// Mitsubishi GX Works2 project: part_B_group31   PLC: FX3G

// global labels: Global1
VAR_GLOBAL
  Ac_start AT X007 : BOOL;
  Ac_stop AT X005 : BOOL;
  Ac_keepOn AT M0 : BOOL;
  one_hour AT TC6 : BOOL;
END_VAR
VAR_GLOBAL CONSTANT
  const_1hour : INT := 60;
END_VAR
VAR_GLOBAL
  one_hour_VAL AT TS6 : BOOL;
  sen_move AT X001 : BOOL;
  Last_move AT M1 : BOOL;
  sen_window AT X002 : BOOL;
  Ac_on AT Y001 : BOOL;
  check_move AT M4 : BOOL;
  Alarm AT Y002 : BOOL;
END_VAR

// task Task_01 (event TRUE, interval 0, priority 31): POU_01

PROGRAM POU_01
(* structured ladder/FBD written out as ST: instructions are called as NAME(EN, inputs, outputs); _pN, _eN, _tN stand for wires *)
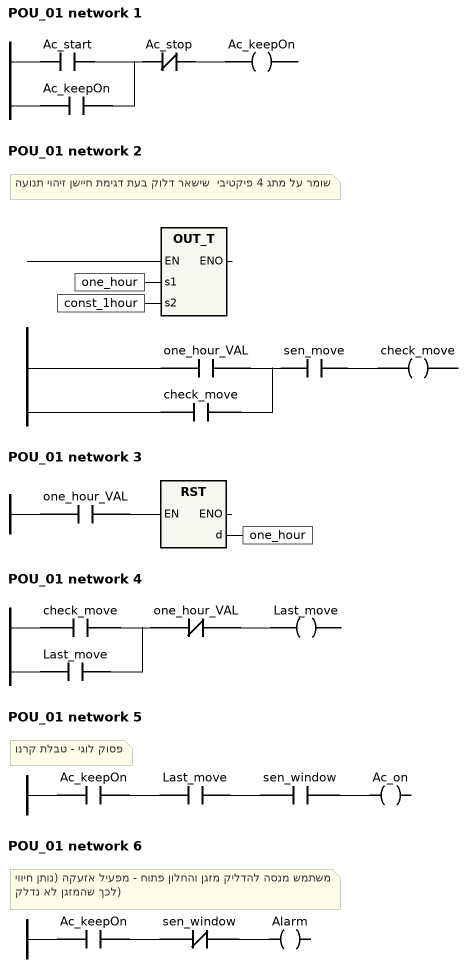
(* network 1 *)
Ac_keepOn := (Ac_start OR Ac_keepOn) AND NOT Ac_stop;
(* network 2 *)
(* שומר על מתג 4 פיקטיבי  שישאר דלוק בעת דגימת חיישן זיהוי תנועה *)
OUT_T(TRUE, one_hour, const_1hour);
check_move := (one_hour_VAL OR check_move) AND sen_move;
(* network 3 *)
RST(one_hour_VAL, one_hour);
(* network 4 *)
Last_move := (check_move OR Last_move) AND NOT one_hour_VAL;
(* network 5 *)
(* פסוק לוגי - טבלת קרנו *)
Ac_on := Ac_keepOn AND Last_move AND sen_window;
(* network 6 *)
(* משתמש מנסה להדליק מזגן והחלון פתוח - מפעיל אזעקה (נותן חיווי (לכך שהמזגן לא נדלק *)
Alarm := Ac_keepOn AND NOT sen_window;
END_PROGRAM
